(* PLC project titulo, CODESYS CODESYS V3.5 SP17 Patch 3, author autor *)
(* stored: creationDateTime 2022-04-22T12:35:31.5064964, version 69.41, modificationDateTime 2022-04-22T11:58:57.9681441, organization compania *)
(* descricao *)

PROGRAM flow1

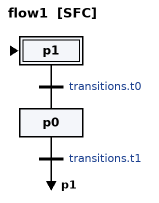
INITIAL_STEP p1:
END_STEP
TRANSITION FROM p1 TO p0
  := transitions.t0;
END_TRANSITION
STEP p0:
END_STEP
TRANSITION FROM p0 TO p1
  := transitions.t1;
END_TRANSITION
END_PROGRAM

PROGRAM flow2

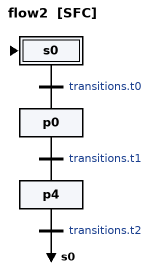
INITIAL_STEP s0:
END_STEP
TRANSITION FROM s0 TO p0
  := transitions.t0;
END_TRANSITION
STEP p0:
END_STEP
TRANSITION FROM p0 TO p4
  := transitions.t1;
END_TRANSITION
STEP p4:
END_STEP
TRANSITION FROM p4 TO s0
  := transitions.t2;
END_TRANSITION
END_PROGRAM

PROGRAM flow4

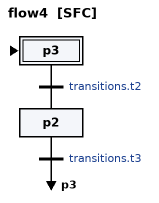
INITIAL_STEP p3:
END_STEP
TRANSITION FROM p3 TO p2
  := transitions.t2;
END_TRANSITION
STEP p2:
END_STEP
TRANSITION FROM p2 TO p3
  := transitions.t3;
END_TRANSITION
END_PROGRAM

PROGRAM flow3

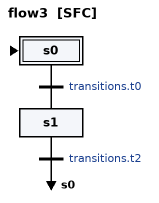
INITIAL_STEP s0:
END_STEP
TRANSITION FROM s0 TO s1
  := transitions.t0;
END_TRANSITION
STEP s1:
END_STEP
TRANSITION FROM s1 TO s0
  := transitions.t2;
END_TRANSITION
END_PROGRAM

PROGRAM transitions

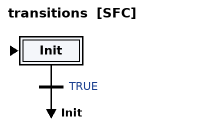
INITIAL_STEP Init:
END_STEP
TRANSITION FROM Init TO Init
  := TRUE;
END_TRANSITION
END_PROGRAM

CONFIGURATION Application
  RESOURCE Application ON PLC
    {attribute 'qualified_only'}
    VAR_GLOBAL  (* GVL *)
      tr0 : BOOL;
      tr1 : BOOL;
      tr2 : BOOL;
      tr3 : BOOL;
    END_VAR
    TASK MainTask(INTERVAL := T#20ms, PRIORITY := 1);
    PROGRAM flow1 WITH MainTask : flow1;
    PROGRAM flow2 WITH MainTask : flow2;
    PROGRAM flow3 WITH MainTask : flow3;
    PROGRAM flow4 WITH MainTask : flow4;
  END_RESOURCE
END_CONFIGURATION
